{attribute 'qualified_only'}
{attribute 'strict'}
TYPE ESequences :
(
	empty := 0,
	sample_sequence := 1
) UINT;
END_TYPE

(* stored: Version 1.1.0.1, ProductVersion 3.1.4024.9
   DUT ESequences: Id {151b3f24-b699-4a41-b19c-ab1e5c6718df} *)
